Fanuc KAREL source: ka00105.KL

-- PROVISIONAL review KL for V1013-1; original PC SHA256 30692e538f399c9eb29844693889eba1259caa8e04f3f4d1b74abdf3c6a8edf1
-- Incomplete behavior may be omitted. Consult companion uncertainty JSON. Do not deploy.
PROGRAM KA00105
%NOLOCKGROUP
-- UNRESOLVED_DECL SRC type=000013
-- UNRESOLVED_DECL DST type=000013
BEGIN
  -- UNRESOLVED_PC offsets 5-20; opcodes 2E,22,32,35
  -- UNRESOLVED_PC offsets 25-40; opcodes 49,4A
  -- UNRESOLVED_PC offsets 45-49; opcodes 7F
END KA00105
